// TwinCAT 3 PLC project PlcElbowControl
// ProgramVersion: 3.1.0.8
// libraries:
//   Tc2_SerialCom, * (Beckhoff Automation GmbH)
//   Tc2_Standard, * (Beckhoff Automation GmbH)
//   Tc2_System, * (Beckhoff Automation GmbH)
//   Tc3_Interfaces, * (Beckhoff Automation GmbH)
//   Tc3_Module, * (Beckhoff Automation GmbH)
// project tree:
//   DUTs/ DATASTRUCT.TcDUT
//   GVLs/ GVL.TcGVL
//   / PlcTask.TcTTO
//   POUs/ Fast.TcPOU (not stored), MAIN.TcPOU, SerialRecieve.TcPOU, WRITEFILE.TcPOU (not stored)
// real-time tasks:
//   TASK PlcTask: cycle T#1ms, priority 20, ADS port 350
//   TASK CppTask: cycle T#1ms, priority 1, ADS port 354
// I/O:
//   DEVICE Device 4 (EtherCAT), AmsNetId 5.39.221.128.5.1
//     Box 1 (CPX-FB37) [CPX-FB37 Fieldbus module]
//       modules: Module 1 (FB37-RIO), Module 1 (VPPM Display 10 bar [1AI/1AO]), Module 1 (VPPM Display 10 bar [1AI/1AO]), Module 1 (VPPM Display 10 bar [1AI/1AO]), Module 1 (VPPM Display 10 bar [1AI/1AO]), Module 1 (VPPM Display 10 bar [1AI/1AO]), Module 1 (VPPM Display 10 bar [1AI/1AO]), Module 1 (VPPM Display 10 bar [1AI/1AO]), Module 1 (VPPM Display 10 bar [1AI/1AO])
//   DEVICE Device 6 (NOV-DP-RAM)
//   DEVICE Device 1 (EtherCAT), AmsNetId 5.39.221.128.2.1
//     Term 1 (EK1200) [EK1200-5000 EtherCAT Power supply (2A E-Bus)]
//       Term 3 (EL2502) [EL2502 2K. PWM Ausgang, 24V]
//       Term 4 (EL6001) [EL6001 Interface (RS232)]
//       Term 5 (EL3002) [EL3002 2Ch. Ana. Input +/-10V]
//       Term 6 (EL4104) [EL4104 4Ch. Ana. Output 0-10V, 16bit]
//       Term 7 (EL4102) [EL4102 2Ch. Ana. Output  0-10V, 16bit]
//       Term 8 (EL3008) [EL3008 8Ch. Ana. Input +/-10V]
//       Term 9 (EL6001) [EL6001 Interface (RS232)]
//       Term 10 (EK1122) [EK1122 2 port EtherCAT junction]
//       Term 11 (EL6002) [EL6002 Interface 2Ch. (RS232)]
//       Term 11 (EL9011) [EL9011 End Terminal]
// variable links:
//   Device 1 (EtherCAT) <-> CppElbowControl/CppElbowControl_Obj1 (CModule1)
//     Term 1 (EK1200)/Term 6 (EL4104)/AO Output Channel 1/Analog output <-> Outputs/m2Int
//     Term 1 (EK1200)/Term 6 (EL4104)/AO Output Channel 2/Analog output <-> Outputs/m1Int
//   PlcElbowControl/PlcElbowControl Instance <-> Device 1 (EtherCAT)/Term 1 (EK1200)/Term 4 (EL6001)
//     PlcTask Inputs/GVL.EL6_22Bin_PC1/D <-> COM Inputs/Data In 0
//     PlcTask Inputs/GVL.EL6_22Bin_PC1/D @bit {8..168 step 8} <-> COM Inputs/Data In {1..21}  (21 links)
//     PlcTask Inputs/GVL.EL6_22Bin_PC1/Status <-> COM Inputs/Status
//     PlcTask Outputs/GVL.EL6_22Bout_PC1/Ctrl <-> COM Outputs/Ctrl
//     PlcTask Outputs/GVL.EL6_22Bout_PC1/D <-> COM Outputs/Data Out 0
//     PlcTask Outputs/GVL.EL6_22Bout_PC1/D @bit {8..168 step 8} <-> COM Outputs/Data Out {1..21}  (21 links)
//   PlcElbowControl/PlcElbowControl Instance <-> Device 4 (EtherCAT)/Box 1 (CPX-FB37)
//     PlcTask Outputs/MAIN.a0 <-> Module 1 (VPPM Display 10 bar [1AI/1AO])/Outputs/Output 0
//     PlcTask Outputs/MAIN.a{1..5} <-> Module 1 (VPPM Display 10 bar [1AI/1AO])/Outputs_{1..5}/Output 0  (5 links)
//   PlcElbowControl/PlcElbowControl Instance <-> CppElbowControl/CppElbowControl_Obj1 (CModule1)
//     PlcTask Inputs/MAIN.m1v <-> Outputs/m1v
//     PlcTask Inputs/MAIN.m2v <-> Outputs/m2v
//     PlcTask Inputs/MAIN.rad <-> Outputs/rad
//     PlcTask Inputs/MAIN.tarrad <-> Outputs/tarrad
//     PlcTask Outputs/GVL.JIAODU <-> Inputs/Angle
//     PlcTask Outputs/MAIN.t <-> Inputs/PlcTimer

CONFIGURATION PlcElbowControl
    RESOURCE PLC ON TwinCAT3
        TASK PlcTask(INTERVAL := T#1ms, PRIORITY := 20);
        PROGRAM WRITEFILE WITH PlcTask : WRITEFILE;
        PROGRAM Fast WITH PlcTask : Fast;
        PROGRAM SerialRecieve WITH PlcTask : SerialRecieve;
        PROGRAM MAIN WITH PlcTask : MAIN;
    END_RESOURCE
END_CONFIGURATION

// ---- DUTs/DATASTRUCT.TcDUT
TYPE DATASTRUCT :
STRUCT
	p1:REAL;
	p2:REAL;
	p3:REAL;
	g:BOOL;
	h:BOOL;
END_STRUCT
END_TYPE

// ---- GVLs/GVL.TcGVL
VAR_GLOBAL
	//读取编码器角度
	EL6_22Bin_PC1	AT %I* 	: KL6inData22b;
	EL6_22Bout_PC1	AT %Q*	: KL6outData22b;
	RxBuffer1: COMBuffer;
	TxBuffer1: COMBuffer;
	JIAODU: REAL;(*单位 度*)
	JIAOSUDU: REAL;(*单位 度*)
	JIAOJIASUDU: REAL;(*单位 度*)
	//往工控机存数据
	DATA :ARRAY[1..200] OF  DATASTRUCT :=[(p1:=0,p2:=0,p2:=0,g:=FALSE,h:=FALSE)];
	bWRITE_TO_FILE:BOOL:=TRUE;
END_VAR

// ---- POUs/SerialRecieve.TcPOU
PROGRAM SerialRecieve
VAR
	i:INT;
    AA:BYTE;
	BB:BYTE;
	RxBufferStep:INT:=0;
    AA_P:BYTE;
	BB_P:BYTE;
	JIAODU_INT:INT;
	J1: REAL:=0;
	J2: REAL:=0;
	J3: REAL:=0;
	W1:REAL:=0;
	W2:REAL:=0;
	t_tip:LREAL:=0.01;
END_VAR

//读取编码器的数值
	IF RxBuffer1.Count<> 0 THEN
		FOR i:=1 TO UINT_TO_INT(RxBuffer1.Count) DO
			IF RxBufferStep=3 THEN
				BB:=RxBuffer1.Buffer[RxBuffer1.RdIdx];
				AA:=AA_P;
				RxBufferStep:=0;
			END_IF
			IF RxBufferStep=2 THEN
				AA_P:=RxBuffer1.Buffer[RxBuffer1.RdIdx];
				RxBufferStep:=3;
			END_IF
			IF RxBufferStep=1 THEN
				IF RxBuffer1.Buffer[RxBuffer1.RdIdx]=90 THEN
					RxBufferStep:=2;
				ELSE
					RxBufferStep:=0;
				END_IF
			END_IF
			IF RxBuffer1.Buffer[RxBuffer1.RdIdx]=165 THEN
				RxBufferStep:=1;
			END_IF

			RxBuffer1.RdIdx:=RxBuffer1.RdIdx+1;
			IF RxBuffer1.RdIdx>300 THEN
				RxBuffer1.RdIdx:=0;
			END_IF
		END_FOR
	RxBuffer1.Count:=0;
	END_IF

	JIAODU_INT:=UINT_TO_INT(AA*256+BB);
	JIAODU:=INT_TO_REAL(JIAODU_INT)*360.0/4096.0;
	J3:=J2;
	J2:=J1;
	J1:=JIAODU;
	JIAOSUDU:=(J1-J2)/t_tip;
	W2:=W1;
	W1:=JIAOSUDU;
	JIAOJIASUDU:=(W1-W2)/t_tip;

END_PROGRAM

// ---- POUs/MAIN.TcPOU
PROGRAM MAIN
VAR
	t AT %Q*: REAL := 0;
	tip : REAL := 0.001;
	tarrad AT %I* : REAL;
	rad AT %I* : REAL;
	m1v AT %I* : REAL;
	m2v AT %I* : REAL;
	err: REAL;
	test AT %Q* : INT;
	a0 AT %Q* : INT;
	a1 AT %Q* : INT;
	a2 AT %Q* : INT;
	a3 AT %Q* : INT;
	a4 AT %Q* : INT;
	a5 AT %Q* : INT;
    N_save: INT := 1;
    ERRORCODE: INT := 0;
	
	v1 AT %I* : INT;
END_VAR

//t := t + tip;
rad;
tarrad;
err := tarrad - rad;
m1v;
m2v;

(*IF  DATA[N_save].g=DATA[N_save].h THEN
		DATA[N_save].p1:=v1;
		DATA[N_save].g:=NOT DATA[N_save].g ;
		N_save:=N_save+1;
		IF  N_save>200 THEN
			N_save:=1;
		END_IF
ELSE
		ERRORCODE:=1;
END_IF*)


IF  DATA[N_save].g=DATA[N_save].h THEN
		DATA[N_save].p1:=tarrad;
		DATA[N_save].p2:=rad;
		DATA[N_save].p3:=err;
		DATA[N_save].p4:=m1v;
		DATA[N_save].p5:=m2v;
		DATA[N_save].g:=NOT DATA[N_save].g ;
		N_save:=N_save+1;
		IF  N_save>200 THEN
			N_save:=1;
		END_IF
ELSE
		ERRORCODE:=1;
END_IF

//IF t<6 THEN
//test := REAL_TO_INT(1*t/6.0*10000);
//a0 := REAL_TO_INT(1*t/6.0*10000);
//a1 := REAL_TO_INT(1*t/6.0*10000);
//a2 := REAL_TO_INT(1*t/6.0*10000);
//a3 := REAL_TO_INT(1*t/6.0*10000);
//a4 := REAL_TO_INT(1*t/6.0*10000);
//a5 := REAL_TO_INT(1*t/6.0*10000);
//END_IF
//IF t>6 AND t<12 THEN
//a4 := REAL_TO_INT(1*(t-6)/6.0*10000);
//END_IF
//IF t>12 AND t<18 THEN
//a1 := REAL_TO_INT(1*(18-t)/6.0*10000);
//a2 := REAL_TO_INT(1*(18-t)/6.0*10000);
//a4 := REAL_TO_INT(1*(18-t)/6.0*10000);
//END_IF

END_PROGRAM
